TYPE ST_Dpad :
STRUCT
	Up: BOOL;
	Down: BOOL;
	Left: BOOL;
	Right: BOOL;
END_STRUCT
END_TYPE

(* stored: Version 1.1.0.1
   DUT ST_Dpad: Id {c497e547-1dfd-4da7-a86e-8ae4d44a7765} *)
